FUNCTION_BLOCK FB_FileHandler
VAR_INPUT
	sNetId: T_AmsNetId;
	sPathName: T_MaxString;
	
END_VAR
VAR_OUTPUT
END_VAR
VAR
	fbFileOpen : FB_FileOpen;
	fbFileClose : FB_FileClose;
	fbFileSeek : FB_FileSeek;
	fbFileTell : FB_FileTell;
	
	
	stepGetFileSize : INT;
	_hFile: UINT;
	
	
END_VAR

fbFileOpen(
	sNetId:= sNetId, 
	sPathName:= sPathName, 
	nMode:= FOPEN_MODEREAD OR FOPEN_MODEPLUS OR FOPEN_MODEBINARY, 
	ePath:= PATH_GENERIC, 
	bExecute:= , 
	tTimeout:= DEFAULT_ADS_TIMEOUT, 
	bBusy=> , 
	bError=> , 
	nErrId=> , 
	hFile=> _hFile);

METHOD GetFileSize : UDINT
VAR_INPUT
END_VAR
CASE stepGetFileSize OF
0:
	





END_CASE
END_METHOD

METHOD Open : BOOL
VAR_INPUT
END_VAR

fbFileOpen(bExecute := TRUE);
IF  NOT fbFileOpen.bBusy AND NOT fbFileOpen.bError THEN
	Open := TRUE;
END_IF
END_METHOD

END_FUNCTION_BLOCK

(* stored: Version 1.1.0.1, ProductVersion 3.1.4024.12
   POU FB_FileHandler: Id {5844bb3c-397e-4aa6-bb38-14333a74bc12}, SpecialFunc None
   Method GetFileSize: Id {e0a81230-20b2-4dc8-866e-ee7755bacd90}
   Method Open: Id {f8827fbf-c071-4a4d-9c9b-c66b86e12f66} *)
